FUNCTION_BLOCK FB_LamparaAsignada_SFC
VAR_INPUT
END_VAR
VAR_OUTPUT
END_VAR
VAR
    Lampara AT %Q*: BOOL;
    Pulsador AT %I*: BOOL;
END_VAR

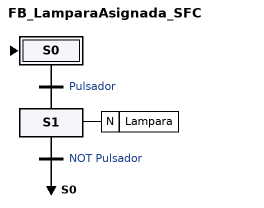
INITIAL_STEP S0:
END_STEP
TRANSITION FROM S0 TO S1
    := Pulsador;
END_TRANSITION
STEP S1:
    Lampara(N);
END_STEP
TRANSITION FROM S1 TO S0
    := NOT Pulsador;
END_TRANSITION

END_FUNCTION_BLOCK

(* stored: Version 1.1.0.1, ProductVersion 3.1.4024.12
   POU FB_LamparaAsignada_SFC: Id {bb4f7988-95ce-42ce-b8e0-58fe48877932}, SpecialFunc None *)
